ABB RobotStudio station: Practica4Entrega.rsstn

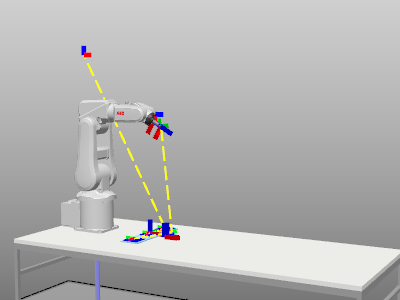
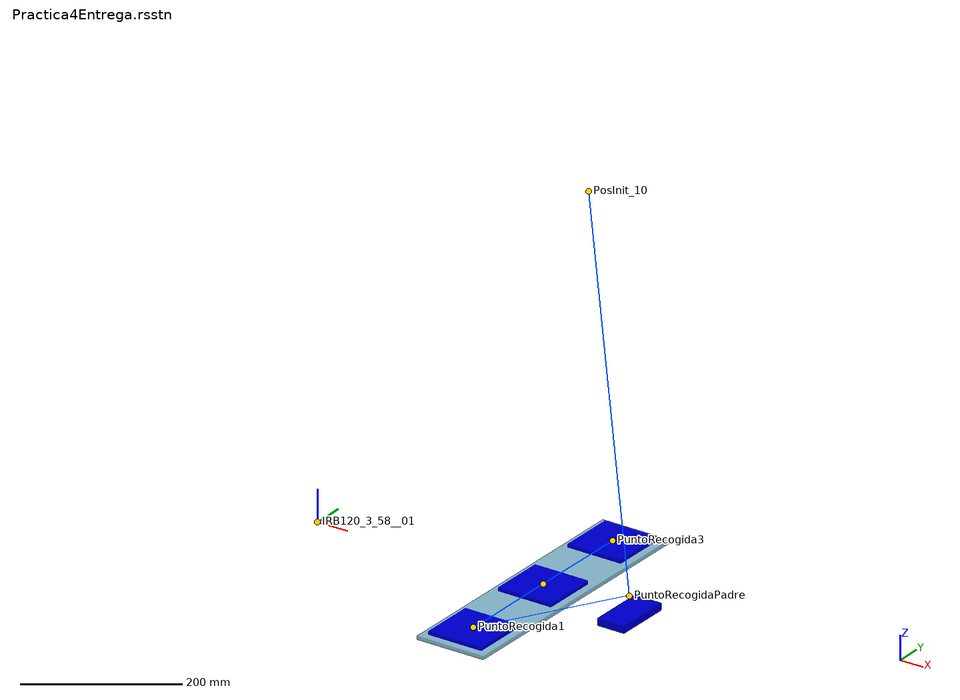
[picture v1: parts stored in the station drawn from their meshes, with robot base, taught points and paths (robot models come from the ABB library and are not in the file)]
Station Práctica3_inicio (saved by RobotStudio 25.1.11133.0)
Controller Controlador2, task T_ROB1: task frame (RAPID world) sits at (0, 0, 670) mm in the station
Controller Controlador2
  mechanical unit ROB_1: IRB120_3_58__01, 6 joints, base frame (0, 0, 0) mm
Layout (positions relative to the parent item):
  - TVentosa [mechanism] at (364.35, 0, 1264) mm, rotated rx 180 ry 60 rz 180 deg
      TCP TVentosa at (0, 0, 51.19) mm
      links: Mi_herramienta
  - LogicGate [smart component, from Components\LogicGate.rslib]
      properties: Operator=NOT; Delay=0
  - LogicGate_2 [smart component, from Components\LogicGate.rslib]
      properties: Operator=AND; Delay=0
  - IRB120_3_58__01 [mechanism, from %ABB.RobotStudio.Models.IRB120%\IRB120_3_58_G_01.rslib] at (0, 0, 670) mm; joint values [0, 0, 0, 0, 0.5236, 0] (rad or m)
  - table [part, from Libraries\e293a11e-ed86-4237-866f-a9bf8f4bd145table.rslib] at (-225, 300, 670) mm, rotated rx 0 ry 0 rz -90 deg
  - SimulationEvents [smart component, from Components\SimulationEvents.rslib]
  - Base0 [part] at (470, 0, 680) mm, size 40 x 80 x 10 mm
  - Base [part], size 100 x 400 x 5 mm
  - Base1 [part], size 80 x 80 x 5 mm
  - Base2 [part], size 80 x 80 x 5 mm
  - Base3 [part], size 80 x 80 x 5 mm
  - Pieza [part] at (470, 0, 680) mm, rotated rx 0 ry 0 rz 90 deg, size 60 x 20 x 20 mm
  - CollisionSensor [smart component, from Components\CollisionSensor.rslib]
      properties: Object1=TVentosa; Object2=(none); NearMiss=0.001; Part1=Mi_herramienta; Part2=(none); CollisionType=1
  - Attacher [smart component, from Components\Attacher.rslib]
      properties: Parent=TVentosa; Flange=0; Child=(none); Mount=false; Offset=[0 0 0]; Orientation=[0 0 0]
  - Detacher [smart component, from Components\Detacher.rslib]
      properties: Child=(none); KeepPosition=true
  - Source [smart component, from Components\Source.rslib]
      properties: Source=Pieza; Copy=(none); Parent=(none); Position=[0.47 0 0.68]; Orientation=[0 0 1.5707963267949]; Transient=false; PhysicsBehavior=-1
Attachment: TVentosa is attached to IRB120_3_58__01 / Link6
Attachment: Base0 is attached to table
Attachment: Base is attached to table
Attachment: Base1 is attached to Base
Attachment: Base2 is attached to Base
Attachment: Base3 is attached to Base
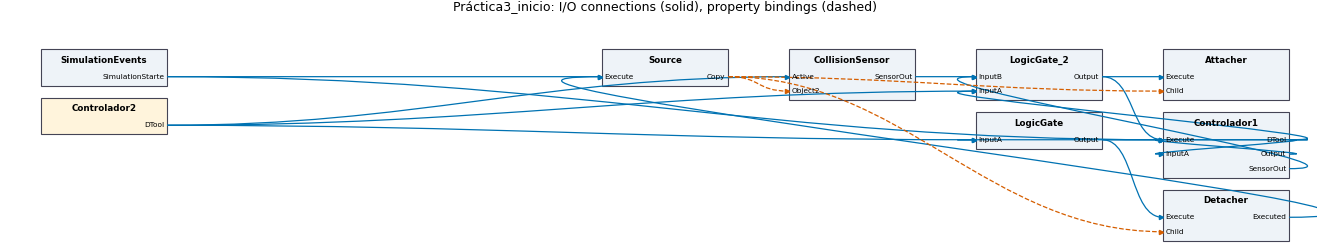
Station logic (signal -> signal, property => property):
  Controlador1.DTool -> Attacher.Execute
  Controlador1.DTool -> LogicGate_2.InputA
  LogicGate_2.Output -> Detacher.Execute
  Controlador1.DTool -> LogicGate.InputA
  LogicGate.Output -> Detacher.Execute
  CollisionSensor.SensorOut -> LogicGate_2.InputB
  Controlador1.DTool -> LogicGate_2.InputA
  LogicGate_2.Output -> Attacher.Execute
  SimulationEvents.SimulationStarted -> Source.Execute
  Controlador2.DTool -> LogicGate_2.InputA
  CollisionSensor.SensorOut -> LogicGate_2.InputB
  LogicGate_2.Output -> Attacher.Execute
  Controlador2.DTool -> LogicGate.InputA
  LogicGate.Output -> Detacher.Execute
  SimulationEvents.SimulationStarted -> Source.Execute
  Detacher.Executed -> Source.Execute
  Controlador2.DTool -> CollisionSensor.Active
  Source.Copy => Attacher.Child
  Source.Copy => Detacher.Child
  Source.Copy => CollisionSensor.Object2
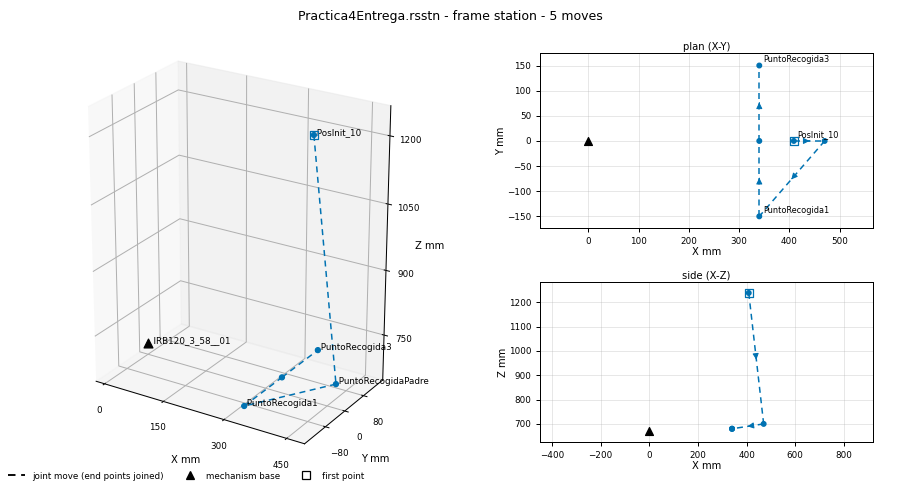
[picture p0: tool path of Practica4Entrega.rsstn in frame station, 5 of 6 moves have a stored position in this frame; points joined in program order, loops and branches not executed]
Targets, tools, work objects and paths stored in the station, written as RAPID:
! task T_ROB1
MODULE CalibData
  PERS tooldata TVentosa:=[TRUE,[[0,0,51.19],[1,0,0,0]],[0.1,[0,0,1],[1,0,0,0],0,0,0]];
  TASK PERS wobjdata WO_Pieza:=[FALSE,TRUE,"",[[450,-40,10],[1,0,0,0]],[[10,10,0],[1,0,0,0]]];
  TASK PERS wobjdata WO_Base:=[FALSE,TRUE,"",[[450,-40,10],[1,0,0,0]],[[-110,40,0],[1,0,0,0]]];
ENDMODULE

! task T_ROB1
MODULE Module1
  CONST robtarget PuntoRecogida1:=[[0,-150,0],[0,-0.707106781,0.707106781,0],[-1,0,-2,0],[9E+09,9E+09,9E+09,9E+09,9E+09,9E+09]];
  CONST robtarget PuntoRecogida2:=[[0,0,0],[0,-0.707106781,0.707106781,0],[0,0,-1,0],[9E+09,9E+09,9E+09,9E+09,9E+09,9E+09]];
  CONST robtarget PuntoRecogida3:=[[0,150,0],[0,-0.707106781,0.707106781,0],[0,0,-1,0],[9E+09,9E+09,9E+09,9E+09,9E+09,9E+09]];
  CONST robtarget PuntoRecogidaPadre:=[[10,30,20],[0,0,1,0],[0,0,0,0],[9E+09,9E+09,9E+09,9E+09,9E+09,9E+09]];
  CONST jointtarget Jhome:=[[0,0,-90,0,0,0],[9E+09,9E+09,9E+09,9E+09,9E+09,9E+09]];
  CONST jointtarget Jcercano:=[[0,0,0,0,0,0],[9E+09,9E+09,9E+09,9E+09,9E+09,9E+09]];
  CONST robtarget PuntoAcercamiento:=[[10,30,50],[0,-0.707106781,0.707106781,0],[0,0,0,0],[9E+09,9E+09,9E+09,9E+09,9E+09,9E+09]];
  CONST robtarget PuntoAcercamiento3:=[[0,150,30],[0,-0.707106781,0.707106781,0],[0,0,-1,0],[9E+09,9E+09,9E+09,9E+09,9E+09,9E+09]];
  CONST robtarget PuntoAcercamiento2:=[[0,0,30],[0,-0.707106781,0.707106781,0],[0,0,-1,0],[9E+09,9E+09,9E+09,9E+09,9E+09,9E+09]];
  CONST robtarget PuntoAcercamiento1:=[[0,-150,30],[0,-0.707106781,0.707106781,0],[-1,0,-2,0],[9E+09,9E+09,9E+09,9E+09,9E+09,9E+09]];
  CONST robtarget PosInit_10:=[[408.685,0,568.405],[0.5,0,0.866025404,0],[0,0,0,0],[9E+09,9E+09,9E+09,9E+09,9E+09,9E+09]];
  CONST jointtarget PosicionInicial:=[[0,-0.000132889,0.000133557,0,30.000000835,0],[9E+09,9E+09,9E+09,9E+09,9E+09,9E+09]];
  PROC Trayectoria()
    MoveJ PosInit_10,v1000,z100,TVentosa\WObj:=wobj0;
    MoveJ PuntoRecogidaPadre,v1000,z100,TVentosa\WObj:=WO_Pieza;
    MoveJ PuntoRecogida1,v1000,z100,TVentosa\WObj:=WO_Base;
    MoveJ PuntoRecogida2,v1000,z100,TVentosa\WObj:=WO_Base;
    MoveJ PuntoRecogida3,v1000,z100,TVentosa\WObj:=WO_Base;
    MoveAbsJ Jhome,v1000,z100,TVentosa\WObj:=wobj0;
  ENDPROC
ENDMODULE

